(* IEC 61131-3 sources: plc_generation_empirical_study/datasets/task_bank_runtime_replacements_v0_1/tasks/C04_M02_toggle_on_edge, 2 files *)

(* ---- interface.st ---- *)
FUNCTION_BLOCK C04_M02_toggle_on_edge
VAR_INPUT
    Button : BOOL;
    Enable : BOOL;
    Reset : BOOL;
END_VAR
VAR_OUTPUT
    State : BOOL;
    AcceptedPulse : BOOL;
END_VAR
END_FUNCTION_BLOCK

(* ---- reference.st ---- *)
FUNCTION_BLOCK C04_M02_toggle_on_edge
VAR_INPUT
    Button : BOOL;
    Enable : BOOL;
    Reset : BOOL;
END_VAR
VAR_OUTPUT
    State : BOOL;
    AcceptedPulse : BOOL;
END_VAR
VAR
    PrevButton : BOOL := FALSE;
END_VAR

AcceptedPulse := FALSE;
IF Reset THEN
    State := FALSE;
ELSIF Enable AND Button AND (NOT PrevButton) THEN
    State := NOT State;
    AcceptedPulse := TRUE;
END_IF;
PrevButton := Button;

END_FUNCTION_BLOCK
